Fanuc KAREL source: kt00403.compact.KL

PROGRAM KT00403
%STACKSIZE=65535
%PRIORITY=65535
%NOLOCKGROUP
VAR
I1 : INTEGER
Y2 : ARRAY[2] OF BYTE
OUT : BOOLEAN
BEGIN
I1=2
Y2[1]=3
OUT=(I1 > Y2[1])
END KT00403
